// TwinCAT 3 PLC project LibraryRfidReaderExample
// Title: Test
// Company: Gema
// Author: RG
// ProjectVersion: 0.1.0.0
// ProgramVersion: 3.1.4023.0
// libraries:
//   RfidReader, * (Gema)
//   Tc2_Standard, * (Beckhoff Automation GmbH)
//   Tc2_System, * (Beckhoff Automation GmbH)
//   Tc3_Module, * (Beckhoff Automation GmbH)
//   TcoCore, 0.11.0.23 (Vortex.Library)
//   TcoData, 0.11.0.23 (Vortex.Library)
//   TcoDrivesBeckhoff, 0.11.0.23 (Vortex.Library)
//   TcoElements, 0.11.0.23 (Vortex.Library)
//   TcoIo, 0.11.0.23 (Vortex.Library)
//   TcoPneumatics, 0.11.0.23 (Vortex.Library)
// project tree:
//   / PlcTask.TcTTO
//   POUs/ AppContext.TcPOU, MAIN.TcPOU (not stored), MainStation.TcPOU
// (motion and I/O tree: see PLC project libraryrfidreader)
// real-time tasks:
//   TASK PlcTask: cycle T#1ms, priority 20, ADS port 350
// variable links:

CONFIGURATION LibraryRfidReaderExample
    RESOURCE PLC ON TwinCAT3
        TASK PlcTask(INTERVAL := T#1ms, PRIORITY := 20);
        PROGRAM MAIN WITH PlcTask : MAIN;
    END_RESOURCE
END_CONFIGURATION

// ---- POUs/AppContext.TcPOU
FUNCTION_BLOCK AppContext EXTENDS TcoCore.TcoContext
VAR
    _mainStation : MainStation(THIS^);

    {attribute addProperty Name "Versionsnummer Plc"}
    _sVersion : STRING(23);
    //~
    _stProgramVersion : ST_LibVersion;
    //~

END_VAR

(*~
    <docu>
        <summary>
            Main method of the TcoContext. This is the entry point of any control logic that belongs to this context.
            The call of this method is ensured by calling the <c>InstanceName.Run()</c> method, and it must not be called explicitly.
            This method is abstract, and it must be overridden in derived block.
        </summary>
    </docu>
~*)
METHOD PROTECTED Main
_mainStation();

//IF (THIS^._startCycleCount MOD 10 = 0) THEN
//    Logger.Push('This is a log entry', eMessageCategory.Trace);
//END_IF;

//IF (THIS^._startCycleCount MOD 125 = 0) THEN
//    Logger.Push('This is a log entry', eMessageCategory.Info);
//END_IF;

//IF (THIS^._startCycleCount MOD 400 = 0) THEN
//    Logger.Push('This is a log entry', eMessageCategory.Warning);
//END_IF;

//IF (THIS^._startCycleCount MOD 2000 = 0) THEN
//    Logger.Push('This is a log entry', eMessageCategory.Error);
//END_IF;
END_METHOD

END_FUNCTION_BLOCK

// ---- POUs/MainStation.TcPOU
FUNCTION_BLOCK MainStation EXTENDS TcoCore.TcoObject
VAR
    counter : INT;
END_VAR

VAR
    compactRfid : RG.Rfid_FB_Compact_Wrapper;
    mockNoRfid : RG.RfidMockNoRfidInRange;
    MockWorking : RG.RfidMockWorking;
    turckRfidHead : RG.RfidHead(THIS^, compactRfid, T#200MS,);
    result : T_MaxString;
    _uid, readData, _reset, _write, _lock : BOOL;

    _isError : BOOL;
    _uiDataRxLength : UINT;
    _uiDataLenght : UINT := 4;
	_startAdress : UINT := 0;
	_length : BYTE := 0;

    _errorId : RG.RFID_FB_U.ERROR;

    _offset : byte;
    _data : ARRAY[0..8] OF BYTE := [0, 2, 4, 6];

    _statusLocked : bool;
END_VAR

//counter := counter + 1;

//IF (THIS^.counter MOD 13 = 0) THEN
//    THIS^.Messenger.Info('opalalla').Pin();
//END_IF

//IF (THIS^.counter MOD 400 = 0) THEN
//    THIS^.Messenger.Error('ich Poste').Pin();
//END_IF

turckRfidHead();
_errorId := turckRfidHead.ErrorId;

IF _uid THEN
    IF turckRfidHead.ReadUidMethod().Error THEN
        _isError := turckRfidHead.IsError;
        _errorId := turckRfidHead.ErrorId;
    ELSIF turckRfidHead.ReadUidMethod().Done THEN
        result := turckRfidHead.Uid;
        _uid   := FALSE;
    END_IF
END_IF

IF _lock THEN
    _statusLocked := FALSE;

    IF turckRfidHead.LockMethod(StartAdress := _startAdress, udiDataLength := _length).Error THEN
        _isError := turckRfidHead.IsError;
        _errorId := turckRfidHead.ErrorId;
    ELSIF turckRfidHead.LockTask.Done THEN
        _lock         := FALSE;
        _statusLocked := TRUE;
    END_IF
END_IF

IF readData THEN
    IF turckRfidHead.ReadDataMethod(_uiDataLenght, _offset).Error THEN
        _isError := turckRfidHead.IsError;
        _errorId := turckRfidHead.ErrorId;
    ELSIF turckRfidHead.ReadDataTask.Done THEN
        _uiDataRxLength := turckRfidHead.DataRxLength;
        readData        := FALSE;
        result          := turckRfidHead.Data;
    END_IF
END_IF

IF _write THEN
    IF turckRfidHead.WriteDataMethod(_data, _offset).Error THEN
        _isError := turckRfidHead.IsError;
        _errorId := turckRfidHead.ErrorId;
    ELSIF turckRfidHead.WriteDataTask.Done THEN
        _uiDataRxLength := turckRfidHead.DataRxLength;
        _write          := FALSE;

    END_IF
END_IF

IF _reset THEN
    _reset := FALSE;
    turckRfidHead.Restore();
    _isError := false;
END_IF

END_FUNCTION_BLOCK
